// TIA Portal V20 export
TYPE "LAxisCtrl_typeDiagnostics"
TITLE = LAxisCtrl_typeDiagnostics
// Support: tech.team.motioncontrol@siemens.com 
// Fax: +49 (0) 9131/98-1297
   STRUCT
      status : Word := 16#0000;   // Status of FB when error occurred
      subfunctionStatus : Word := 16#0000;   // ErrorID of called subfunction
      basicMotionState : DInt := 0;   // Current basic motion state when error occurred
      superimposedMotionState : DInt := 0;   // Current superimposed motion state when error occurred
   END_STRUCT;
END_TYPE
